FUNCTION LinTrafoLimitLess : REAL
VAR_INPUT
	rValue:REAL;			(*Valor a sofrer escala*)
	rInMin:REAL;			(*Valor minimo de entrada*)
	rInMax:REAL;			(*valor Maximo de entrada*)
	rOutMin:REAL;		(*Valor minimo da saida*)
	rOutMax:REAL;		(*Valor maximo de saida*)
END_VAR
VAR
END_VAR
(*Esta funcao admite tanto valores negativos quanto positivos (porem a saida so sera negativa se o valor de entrada for negativo)*)

(*Realiza uma simples escala*)
LinTrafoLimitLess:=rValue*(rOutMax-rOutMin)/CheckDivZero(rInMax-rInMin);

END_FUNCTION

(* stored: Version 1.1.0.1, ProductVersion 3.1.4024.12
   POU LinTrafoLimitLess: Id {d0ca79a4-037c-47d1-8f3e-1712e918b4a5}, SpecialFunc None *)
